// This function has been automatically generated from the project information.
{attribute 'signature_flag' := '1073741824'}
{attribute 'TcGenerated'}
{attribute 'no-analysis'}
FUNCTION F_GetCompany : WSTRING
VAR_INPUT
	
END_VAR

F_GetCompany := "Gauggel";

END_FUNCTION

(* stored: Version 1.1.0.1
   POU F_GetCompany: Id {d725d5a3-2093-4c8b-a014-b3fd51cf2299}, SpecialFunc None *)
